
FUNCTION CB_dword_to_byte : BYTE

TITLE = ' Convert a double word into a byte '
VERSION : '1.0'
AUTHOR  : CB
NAME    : DintToBy
FAMILY  : TNI

VAR_INPUT
    IN : DWORD;
END_VAR

VAR_TEMP

END_VAR

BEGIN

CB_dword_to_byte := DWORD_TO_BYTE(IN);

END_FUNCTION
